// TIA Portal V16 export
// export: Created 2021-09-03T13:57:09.0792558Z, ExportSetting WithDefaults, DisplayName Totally Integrated Automation Portal, DisplayVersion V16 Update 3, DisplayName TIA Portal Version Control Interface, DisplayVersion V16 Update 2, DisplayName TIA Portal Openness, DisplayVersion V16 Update 3, DisplayName TIA Portal Teamcenter Gateway, DisplayVersion V16, DisplayName STEP 7 Professional, DisplayVersion V16 Update 3, DisplayName STEP 7 Safety, DisplayVersion V16, DisplayName WinCC Advanced, DisplayVersion V16 Update 3
TYPE "UF_PARAMETRS"
// stored: IsFailsafeCompliant false
   STRUCT
      valueHDP : Real;
      delayHDP : UInt;
      countHWbyHDP : UInt;
      maxNumbHWbyHDP : UInt;
   END_STRUCT;
END_TYPE
